# EPICS substitutions: TPG300/TPG300-IOC-01App/Db/unit_setter.substitutions
# Set points do not have units set because it will cause it to be processed thus sending a possibly wrong value
# to the display

file $(UTILITIES)/db/unit_setter.template {
  pattern
    {P,    FROM, TO}

    {"\$(P)", "UNITS", "PRESSURE_A1"}
    {"\$(P)", "UNITS", "PRESSURE_A2"}
    {"\$(P)", "UNITS", "PRESSURE_B1"}
	{"\$(P)", "UNITS", "PRESSURE_B2"}
}
